// SIMATIC S7-200 project (STEP 7-Micro/WIN), CPU 222 REL 01.22

SYMBOL_TABLE USR1
程序启动             I0.0
程序停止             I0.1
整定脉宽1            I0.2
整定脉宽2            I0.3
提升阀1运行           Q0.0
提升阀2运行           Q0.1
提升阀3运行           Q0.2
提升阀4运行           Q0.3
提升阀5运行           Q0.4
提升阀6运行           Q0.5
脉冲阀1运行           Q1.0
脉冲阀2运行           Q1.1
脉冲阀3运行           Q1.2
脉冲阀4运行           Q1.3
脉冲阀5运行           Q1.4
脉冲阀6运行           Q1.5
程序运行指示           Q1.6
END_SYMBOL_TABLE

ORGANIZATION_BLOCK MAIN:OB1
TITLE=运行当前程序的PLC设备放在立窑生料磨生产线的收尘器控制系统中。负责管理六个提升阀和脉冲阀的运行。经过现实应用，情况表现良好，没发现有什么问题。
// 系统启动时，首先根据脉宽选择开关1和脉宽选择开关2的状态设置脉冲阀的运行时间，时间只能在12、15或20中选择。如果两个开关都未按下，脉宽默认为12；若按下脉宽选择开关1，则设为15；若按下脉宽选择开关2，则设为20。这一设置决定了后续脉冲阀喷吹的时长。
// 当内部标志为真时，程序运行指示灯点亮，表示清灰程序正式运行，此时系统开始协调提升阀和脉冲阀的工作。
// 每当T37到时，计数器C0递增一次，从1到6，依次决定当前激活的提升阀。
// 计数器C0的递增仅在T37到时且程序运行指示灯为真时发生，最大值固定为6，确保清灰循环不会超出预定范围。
// 当计数器C0值为1且内部标志为真时，激活另一内部标志。
// 当该内部标志为真时，打开提升阀1控制。
// 当提升阀运行时，T37定时器启动。
// 当T37为真时，T35定时器启动并触发脉冲阀1控制喷吹，完成第一组滤袋的清灰。
// 脉冲阀1控制只有在提升阀1控制运行且T35激活时才会工作。
// 当计数器C0增至2至6时，分别激活对应的内部标志。
// 当这些内部标志为真时，依次激活提升阀2控制至提升阀6控制及其对应的脉冲阀2控制至脉冲阀6控制，完成后续滤袋清灰。
// 
BEGIN
Network 1
LD     SM0.0
LPS
AN     整定脉宽1:I0.2
AN     整定脉宽2:I0.3
MOVW   +12, VW100
LRD
A      整定脉宽1:I0.2
MOVW   +15, VW100
LPP
A      整定脉宽2:I0.3
MOVW   +20, VW100
Network 2
LD     M0.0
=      程序运行指示:Q1.6
Network 3
LD     SM0.0
LPS
BTI    SMB28, AC0
*I     +12, AC0
+I     +100, AC0
AW>=   AC0, +3000
MOVW   +3000, AC0
LPP
MOVW   AC0, VW100
Network 4
LD     M0.0
AN     T37
TON    T37, VW100
Network 5
LD     程序运行指示:Q1.6
A      T37
LD     C0
CTU    C0, +6
Network 6
LD     M0.0
LPS
AW=    C0, +1
=      M0.1
LRD
AW=    C0, +2
=      M0.2
LRD
AW=    C0, +3
=      M0.3
LRD
AW=    C0, +4
=      M0.4
LRD
AW=    C0, +5
=      M0.5
LPP
AW=    C0, +6
=      M0.6
Network 7
LD     M0.1
O      M0.2
O      M0.3
O      M0.4
O      M0.5
O      M0.6
AN     T37
TON    T37, +20
Network 8
LD     T37
TOF    T35, VW100
Network 9
LD     M0.1
=      提升阀1运行:Q0.0
A      T35
=      脉冲阀1运行:Q1.0
Network 10
LD     M0.2
=      提升阀2运行:Q0.1
A      T35
=      脉冲阀2运行:Q1.1
Network 11
LD     M0.3
=      提升阀3运行:Q0.2
A      T35
=      脉冲阀3运行:Q1.2
Network 12
LD     M0.4
=      提升阀4运行:Q0.3
A      T35
=      脉冲阀4运行:Q1.3
Network 13
LD     M0.5
=      提升阀5运行:Q0.4
A      T35
=      脉冲阀5运行:Q1.4
Network 14
LD     M0.6
=      提升阀6运行:Q0.5
A      T35
=      脉冲阀6运行:Q1.5
END_ORGANIZATION_BLOCK
